FUNCTION_BLOCK "Syntax_MissingEndVar"
{ S7_Optimized_Access := 'TRUE' }
VERSION : 0.1

VAR
    value : Int;

BEGIN
    // EXPECT: error[syntax.expected-end-var] SYN-DECL-003
    #value := 1;
END_FUNCTION_BLOCK
